(* PLC project v0.6.04_CycleSemiAuto.project, CODESYS CODESYS V3.5 SP19 Patch 1 *)
(* stored: creationDateTime 2026-08-04T10:25:40.640256, modificationDateTime 2026-08-04T10:25:40.640256 *)

(* ═══════════════════════════════════════════════════════════════ 📡 ST_NetworkDiagHMI — Données d'échange IHM pour les diagnostics réseau ─────────────────────────────────────────────────────────────── 🎨 Destiné à l'affichage des diagnostics CANopen et EtherCAT. ═══════════════════════════════════════════════════════════════ *)
TYPE ST_NetworkDiagHMI : STRUCT
  BusCanOpen : ST_Diag_Device;  (* 📡 Diagnostics bus CANopen *)
  Joystick : ST_Diag_Device;  (* 🕹️ Diagnostics esclave Joystick *)
  CanError : BOOL;  (* ⚠️ Anomalie CANopen *)
  CanErrorId : WORD;  (* ❌ Code anomalie CANopen *)
  BusEthercat : ST_Diag_Device;  (* 📡 Diagnostics bus EtherCAT *)
  EncoderM1 : ST_Diag_Device;  (* 🧲 Diagnostics esclave COD1 *)
  EncoderM2 : ST_Diag_Device;  (* 🧲 Diagnostics esclave COD2 *)
  VariateurM3 : ST_Diag_Device;  (* ↔️ Diagnostics esclave AC600 *)
  EcatError : BOOL;  (* ⚠️ Anomalie EtherCAT *)
  EcatErrorId : WORD;  (* ❌ Code anomalie EtherCAT *)
  InputModules : ST_InputModuleDiagHMI;  (* 🩺 Diagnostic carte des 3 modules DI TOR réelles *)
  Bypass : ST_BypassNetwork;  (* 🌐 Bypass réseau global *)
END_STRUCT;
END_TYPE

(* ═══════════════════════════════════════════════════════════════ 🌐 ST_BypassNetwork — Bypass général du diagnostic réseau ─────────────────────────────────────────────────────────────── 🔒 Permet de forcer les esclaves réseau (CAN, EtherCAT) à "online" pour le diagnostic, sans devoir toucher à chaque bit individuel. Jamais actif en production. ═══════════════════════════════════════════════════════════════ *)
TYPE ST_BypassNetwork : STRUCT
  Joystick : BOOL;  (* 📡 1. Communication & Systèmes esclaves 🕹️ Bypass diagnostic esclave CANopen Joystick *)
  EncoderM1 : BOOL;  (* 🧲 Bypass diagnostic esclave EtherCAT COD1 (M1 codeur) *)
  EncoderM2 : BOOL;  (* 🧲 Bypass diagnostic esclave EtherCAT COD2 (M2 codeur) *)
  VariateurM3 : BOOL;  (* ↔️ Bypass diagnostic esclave EtherCAT AC600 (M3 drive) *)
  IhmHeartbeat : BOOL := TRUE;  (* 💓 Bypass du bit de vie IHM (défaut TRUE = sécurisé si pas d'IHM) *)
  Global : BOOL;  (* 🛡️ 2. Hiérarchie & Restauration 🌐 Bypass Global : tous les esclaves réseau à la fois *)
  Initialized : BOOL := FALSE;  (* 🐛 FIX persistance (voir DOC/AUDITS/ConfigPersistence/) : flag restauration boot dédié (défaut FALSE non ambigu, contrairement à une valeur métier) — PRG_SUPERVISION_CFC.st 🚦 TRUE = bypass restauré depuis GVL_BypassRetain ce boot *)
END_STRUCT;
END_TYPE

(* ═══════════════════════════════════════════════════════════════ 📡 ST_Diag_Device — Structure diagnostic d'un esclave ou bus ═══════════════════════════════════════════════════════════════ *)
TYPE ST_Diag_Device : STRUCT
  Online : BOOL;  (* Esclave visible sur le bus *)
  Operational : BOOL;  (* Esclave en mode OP (opérationnel) *)
  Error : BOOL;  (* Signal de défaut actif pour cet esclave *)
  ErrorId : WORD;  (* Code défaut détaillé *)
  State : E_Diag_State;  (* Phase courante du cycle de diagnostic *)
  StateAtError : E_Diag_State;  (* Instantané de la phase lors de l'anomalie *)
END_STRUCT;
END_TYPE

(* ═══════════════════════════════════════════════════════════════ 🩺 ST_InputModuleDiagHMI — Diagnostic carte des modules DI TOR réelles ─────────────────────────────────────────────────────────────── 📄 Doc métier : DOC/AF/AF_Partie-06_Acquisition_Qualification_IO_v2.3.md §3bis 🎨 Granularité MODULE (pas canal) : GetDeviceState() est un état de carte, pas un diagnostic par voie. Un module en défaut ne dit pas *quelle* TOR ment, seulement qu'aucune des TOR qu'il porte n'est fiable. 🔗 Producteur : PRG_02_Acquisition (3 appels GetDeviceState()). ═══════════════════════════════════════════════════════════════ *)
TYPE ST_InputModuleDiagHMI : STRUCT
  LocalDigitalIoOk : BOOL;  (* TRUE = module Local_Digital_IO opérationnel (8 TOR Winch/Machine) *)
  Vh0800EndOk : BOOL;  (* TRUE = module VH_0800END opérationnel (7 TOR freins/thermiques/AU) *)
  Vh0808EtpOk : BOOL;  (* TRUE = module VH_0808ETP opérationnel (7 TOR positions M3/hydraulique/crible) *)
  Fault : BOOL;  (* TRUE = au moins un des 3 modules DI hors service *)
END_STRUCT;
END_TYPE

(* values of E_Diag_State: DISABLED: Désactivé (surveillance non active); READY: Opérationnel réel, pas de défaut; INIT: Initialisation / Recherche de réseau; MONITORING: Surveillance active (états transitoires); ERROR: Anomalie de communication; SIMULATED: Bypass simulation ou bypass réseau IHM — pas le bus réel *)

{attribute 'qualified_only'}
{attribute 'strict'}
TYPE E_Diag_State : (DISABLED := 0, READY := 1, INIT := 2, MONITORING := 3, ERROR := 4, SIMULATED := 5);
END_TYPE
